// TIA Portal project "2022.06.04_计数器" (V17)

(* hardware
DEVICE "S7-1200 station_1"  S7-1200 Station
   slot 0: "Rack_0"  S7-1200 Rack  Rack  V1.0
   slot 1: "PLC_1"  CPU 1212C DC/DC/DC  6ES7 212-1AE40-0XB0  V4.5
*)

// ===== PLC "PLC_1"  CPU 1212C DC/DC/DC =====

VAR_GLOBAL   // PLC tag table "默认变量表"
   "Tag_1" AT %I0.0 : Bool;
   "自动复位" AT %M0.0 : Bool;
   "Tag_3" AT %I0.2 : Bool;
   "Tag_4" AT %MW10 : Int;
   "Tag_5" AT %Q0.0 : Bool;
   "手动复位" AT %I0.1 : Bool;
   "初始位" AT %M1.0 : Bool;
   "Tag_2" AT %M0.1 : Bool;
   "赋值" AT %I0.3 : Bool;
   "Tag_7" AT %I0.4 : Bool;
   "加" AT %I0.5 : Bool;
   "Tag_9" AT %M10.0 : Bool;
   "减" AT %I0.6 : Bool;
   "手动复位(1)" AT %I0.7 : Bool;
   "Tag_12" AT %M10.1 : Bool;
   "当前值" AT %MW20 : Int;
END_VAR

// folder: System blocks/Program resources

DATA_BLOCK "IEC_Counter_0_DB"   // DB1
{ S7_Optimized_Access := 'TRUE' }
AUTHOR : Simatic
FAMILY : IEC
NAME : CNTR
VERSION : 1.0
// stored: InstanceOfName IEC_COUNTER
"IEC_COUNTER"
BEGIN
END_DATA_BLOCK

DATA_BLOCK "IEC_Counter_0_DB_1"   // DB2
{ S7_Optimized_Access := 'TRUE' }
AUTHOR : Simatic
FAMILY : IEC
NAME : CNTR
VERSION : 1.0
// stored: InstanceOfName IEC_COUNTER
"IEC_COUNTER"
BEGIN
END_DATA_BLOCK

DATA_BLOCK "IEC_Counter_0_DB_2"   // DB3
{ S7_Optimized_Access := 'TRUE' }
AUTHOR : Simatic
FAMILY : IEC
NAME : CNTR
VERSION : 1.0
// stored: InstanceOfName IEC_COUNTER
"IEC_COUNTER"
BEGIN
END_DATA_BLOCK

// folder: (top level)

ORGANIZATION_BLOCK "Main"   // OB1, LAD, ProgramCycle
TITLE = "Main Program Sweep (Cycle)"
{ S7_Optimized_Access := 'TRUE' }
VERSION : 0.1
   VAR_INPUT
      Initial_Call : Bool;   // Initial call of this OB
      Remanence : Bool;   // =True, if remanent data are available
   END_VAR
BEGIN

REGION Network 1
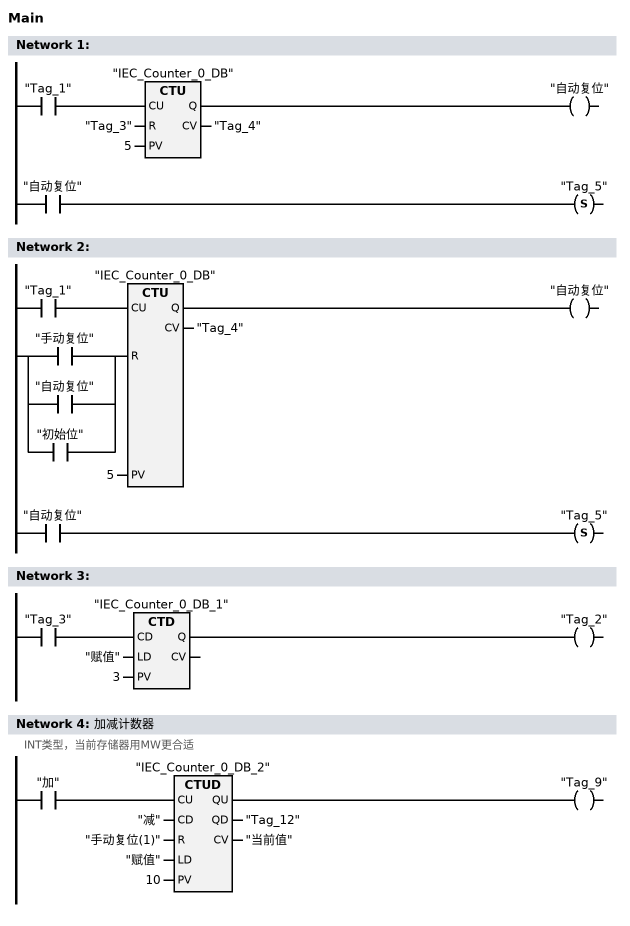
   "IEC_Counter_0_DB".CTU(CU := "Tag_1", R := "Tag_3", PV := 5, CV => "Tag_4");
   "自动复位" := "IEC_Counter_0_DB".Q;
   IF "自动复位" THEN "Tag_5" := TRUE; END_IF;
END_REGION

REGION Network 2
   "IEC_Counter_0_DB".CTU(CU := "Tag_1", R := "手动复位" OR "自动复位" OR "初始位", PV := 5, CV => "Tag_4");
   "自动复位" := "IEC_Counter_0_DB".Q;
   IF "自动复位" THEN "Tag_5" := TRUE; END_IF;
END_REGION

REGION Network 3
   "IEC_Counter_0_DB_1".CTD(CD := "Tag_3", LD := "赋值", PV := 3);
   "Tag_2" := "IEC_Counter_0_DB_1".Q;
END_REGION

REGION Network 4: 加减计数器
   // INT类型，当前存储器用MW更合适
   "IEC_Counter_0_DB_2".CTUD(CU := "加",
                           CD := "减",
                           R := "手动复位(1)",
                           LD := "赋值",
                           PV := 10,
                           QD => "Tag_12",
                           CV => "当前值");
   "Tag_9" := "IEC_Counter_0_DB_2".QU;
END_REGION
END_ORGANIZATION_BLOCK